///EL2252 | XFC, 2-channel digital output terminal with time stamp, tri-state
FUNCTION_BLOCK EL2252_v0_00

END_FUNCTION_BLOCK

(* stored: Version 1.1.0.1, ProductVersion 3.1.0.25
   POU EL2252_v0_00: Id {1cc9bdce-6ea8-4421-a606-54f74ba031be} *)
